{attribute 'qualified_only'}
{attribute 'to_string'}
TYPE E_TimeInstanceKind :
(
	_ := 0, // Uninitialised or default value, indicating an undefined time instance kind.
	UTC,  // The time instance is in Coordinated Universal Time (UTC).
	Local // The time instance is in local time.
);
END_TYPE

(* stored: Version 1.1.0.1
   EnumerationTextList E_TimeInstanceKind: Id {237b53f1-15c5-04ad-378c-7a724cd9e29e} *)
